FUNCTION_BLOCK FB_WordsToFloat32MLE
////////////////// 
// Merge two words or one word into a Real with Mid little endian coding.
//Validée par KBT : 8/11/2017 
//////////////////		
VAR_INPUT
	
	InFirstWord AT %MW0: WORD; 		// Word sent or stored first 
	InSecondWord AT %MW1 : WORD; 	// Word sent or stored last  

END_VAR
VAR_OUTPUT
	OutCalReal AT %MD0 : REAL;		//Output : Real
END_VAR

END_FUNCTION_BLOCK

(* stored: Version 1.1.0.1, ProductVersion 3.1.4024.6
   POU FB_WordsToFloat32MLE: Id {96f5be73-1d99-466a-ba97-5b335ef5f200}, SpecialFunc None *)
